(* IEC 61131-3 sources: programs/VI-54/VI-54_20171205/VI-54_20171205/Stations/Screen/LseClass170718/Class/test, 1 file *)

(* ---- test.st ---- *)
(*!
<Class
	Name               = "test"
	Revision           = "0.0"
	RealtimeTask       = "false"
	CyclicTask         = "true"
	BackgroundTask     = "false"
	Sigmatek           = "false"
	OSInterface        = "false"
	HighPriority       = "false"
	Automatic          = "false"
	UpdateMode         = "Prescan"
	SharedCommandTable = "true"
	Objectsize         = "(284,120)">
	<Channels>
		<Server Name="ClassSvr" Visualized="false" Initialize="false" WriteProtected="false" Retentive="false"/>
		<Server Name="Test2" Visualized="false" Initialize="false" WriteProtected="true" Retentive="false"/>
		<Server Name="Test3" Visualized="false" Initialize="false" WriteProtected="true" Retentive="false"/>
		<Client Name="input2" Required="false" Internal="false"/>
	</Channels>
</Class>
*)
test : CLASS
  //Servers:
	ClassSvr 	: SvrChCmd_DINT;
	Test2 	: SvrCh_DINT;
	Test3 	: SvrCh_DINT;
  //Clients:
	input2 	: CltCh_DINT;
  //Variables:
  //Functions:

	FUNCTION VIRTUAL GLOBAL CyWork
		VAR_INPUT
			EAX 	: UDINT;
		END_VAR
		VAR_OUTPUT
			state (EAX) 	: UDINT;
		END_VAR;
  //Tables:
	FUNCTION @STD
		VAR_OUTPUT
			ret_code	: CONFSTATES;
		END_VAR;
	FUNCTION GLOBAL TAB @CT_;
END_CLASS;

FUNCTION VIRTUAL GLOBAL test::CyWork
	VAR_INPUT
		EAX 	: UDINT;
	END_VAR
	VAR_OUTPUT
		state (EAX) 	: UDINT;
	END_VAR

  input2 := input2.Read();

  // Lezen
  if input2 = 1 then
    TEST3 := 4;
  else
    Test3 := 0;
  end_if;

  Test2 := ClassSvr;

	state := READY;

END_FUNCTION
